KUKA KRL program: ho_lca_st03_pos03.src, ho_lca_st03_pos03.dat

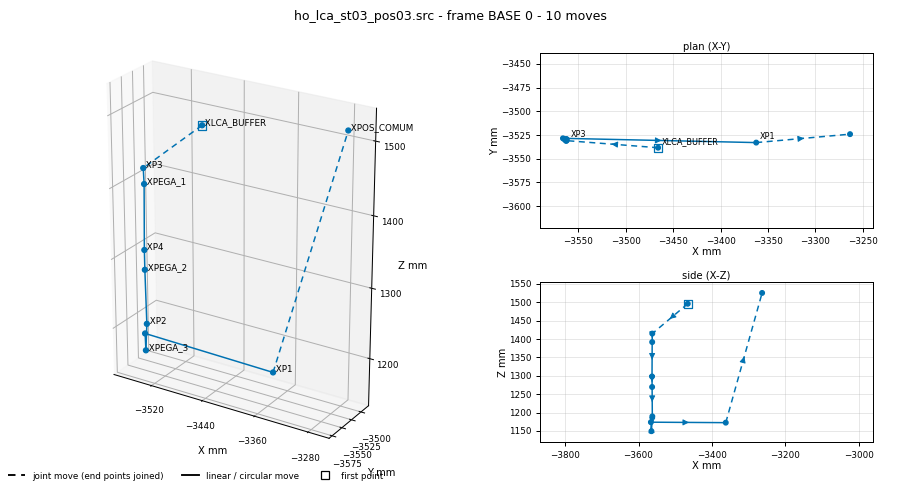
[picture p0: tool path of ho_lca_st03_pos03.src in frame BASE 0, 10 of 10 moves have a stored position in this frame; points joined in program order, loops and branches not executed]
--- ho_lca_st03_pos03.src ---
&ACCESS RVP7
&REL 14
&COMMENT POS_3 LCA
&PARAM DISKPATH = KRC:\R1\Program\LCA
&PARAM TEMPLATE = C:\KRC\Roboter\Template\vorgabe
&PARAM EDITMASK = *
DEF ho_lca_st03_pos03( )
;FOLD INI
  ;FOLD BASISTECH INI
    GLOBAL INTERRUPT DECL 3 WHEN $STOPMESS==TRUE DO IR_STOPM ( )
    INTERRUPT ON 3
    BAS (#INITMOV,0 )
  ;ENDFOLD (BASISTECH INI)
;FOLD SPOTTECH INI
USERSPOT(#INIT)
;ENDFOLD (SPOTTECH INI)
;FOLD GRIPPERTECH INI
USER_GRP(0,DUMMY,DUMMY,GDEFAULT)
;ENDFOLD (GRIPPERTECH INI)
  ;FOLD USER INI
    ;Make your modifications here

  ;ENDFOLD (USER INI)
;ENDFOLD (INI)

; Caracterizacao dos meios de producao
; Changes: Pega LCA Posicao 3 (Pc 3)
; Versao Atual:05/01/2016
; Name: P13.050-R2

chk_w7_wechs_ok ( )   ; CHECK GRIPPER AXOR/ATEGO

;FOLD PTP LCA_BUFFER Vel=100 % DEFAULT Tool[15]:AUX. LCA Base[0];%{PE}%R 8.2.20,%MKUKATPBASIS,%CMOVE,%VPTP,%P 1:PTP, 2:LCA_BUFFER, 3:, 5:100, 7:DEFAULT
$BWDSTART=FALSE
PDAT_ACT=PDEFAULT
FDAT_ACT=FLCA_BUFFER
BAS(#PTP_PARAMS,100)
PTP XLCA_BUFFER
;ENDFOLD

;FOLD WAIT FOR ( IN 3362 'Lib. Pega LCA pos. 3 Axor/Atego' );%{PE}%R 8.2.20,%MKUKATPBASIS,%CEXT_WAIT_FOR,%VEXT_WAIT_FOR,%P 2:, 4:, 5:$IN, 6:3362, 7:Lib. Pega LCA pos. 3 Axor/Atego, 9:
WAIT FOR  ( $IN[3362] )
;ENDFOLD

;FOLD PTP P3 Vel=100 % PDAT1 Tool[15]:AUX. LCA Base[0];%{PE}%R 8.2.20,%MKUKATPBASIS,%CMOVE,%VPTP,%P 1:PTP, 2:P3, 3:, 5:100, 7:PDAT1
$BWDSTART=FALSE
PDAT_ACT=PPDAT1
FDAT_ACT=FP3
BAS(#PTP_PARAMS,100)
PTP XP3
;ENDFOLD

;FOLD WAIT FOR ( NOT IN 489 'Presença pç 1 - Axor LCA' );%{PE}%R 8.2.20,%MKUKATPBASIS,%CEXT_WAIT_FOR,%VEXT_WAIT_FOR,%P 2:, 4:NOT, 5:$IN, 6:489, 7:Presença pç 1 - Axor LCA, 9:
WAIT FOR  (  NOT $IN[489] )
;ENDFOLD

;FOLD ; POSIÇÃO 1 LCA AUSENTE;%{PE}%R 8.2.20,%MKUKATPBASIS,%CCOMMENT,%VNORMAL,%P 2:POSIÇÃO  1 LCA  AUSENTE
;ENDFOLD
;FOLD LIN PEGA_1 Vel=0.1 m/s L_OLP8 Tool[15]:AUX. LCA Base[0];%{PE}%R 8.2.20,%MKUKATPBASIS,%CMOVE,%VLIN,%P 1:LIN, 2:PEGA_1, 3:, 5:0.1, 7:L_OLP8
$BWDSTART=FALSE
LDAT_ACT=LL_OLP8
FDAT_ACT=FPEGA_1
BAS(#CP_PARAMS,0.1)
LIN XPEGA_1
;ENDFOLD

;FOLD LIN P4 Vel=0.05 m/s CPDAT3 Tool[15]:AUX. LCA Base[0];%{PE}%R 8.2.20,%MKUKATPBASIS,%CMOVE,%VLIN,%P 1:LIN, 2:P4, 3:, 5:0.05, 7:CPDAT3
$BWDSTART=FALSE
LDAT_ACT=LCPDAT3
FDAT_ACT=FP4
BAS(#CP_PARAMS,0.05)
LIN XP4
;ENDFOLD

;FOLD WAIT FOR ( NOT IN 489 'Presença pç 1 - Axor LCA' );%{PE}%R 8.2.20,%MKUKATPBASIS,%CEXT_WAIT_FOR,%VEXT_WAIT_FOR,%P 2:, 4:NOT, 5:$IN, 6:489, 7:Presença pç 1 - Axor LCA, 9:
WAIT FOR  (  NOT $IN[489] )
;ENDFOLD

;FOLD ; POSIÇÃO 2 LCA AUSENTE;%{PE}%R 8.2.20,%MKUKATPBASIS,%CCOMMENT,%VNORMAL,%P 2:POSIÇÃO  2 LCA  AUSENTE
;ENDFOLD
;FOLD LIN PEGA_2 Vel=0.05 m/s L_OLP7 Tool[15]:AUX. LCA Base[0];%{PE}%R 8.2.20,%MKUKATPBASIS,%CMOVE,%VLIN,%P 1:LIN, 2:PEGA_2, 3:, 5:0.05, 7:L_OLP7
$BWDSTART=FALSE
LDAT_ACT=LL_OLP7
FDAT_ACT=FPEGA_2
BAS(#CP_PARAMS,0.05)
LIN XPEGA_2
;ENDFOLD

;FOLD LIN P2 Vel=0.05 m/s CPDAT2 Tool[15]:AUX. LCA Base[0];%{PE}%R 8.2.20,%MKUKATPBASIS,%CMOVE,%VLIN,%P 1:LIN, 2:P2, 3:, 5:0.05, 7:CPDAT2
$BWDSTART=FALSE
LDAT_ACT=LCPDAT2
FDAT_ACT=FP2
BAS(#CP_PARAMS,0.05)
LIN XP2
;ENDFOLD

;FOLD ; POSIÇÃO 3 DE PEGA DA PEÇA;%{PE}%R 8.2.20,%MKUKATPBASIS,%CCOMMENT,%VNORMAL,%P 2:POSIÇÃO  3 DE PEGA DA PEÇA
;ENDFOLD
;FOLD LIN PEGA_3 Vel=0.05 m/s L_OLP5 Tool[15]:AUX. LCA Base[0];%{PE}%R 8.2.20,%MKUKATPBASIS,%CMOVE,%VLIN,%P 1:LIN, 2:PEGA_3, 3:, 5:0.05, 7:L_OLP5
$BWDSTART=FALSE
LDAT_ACT=LL_OLP5
FDAT_ACT=FPEGA_3
BAS(#CP_PARAMS,0.05)
LIN XPEGA_3
;ENDFOLD

IF (NOT(GHOST())) THEN
;FOLD WAIT FOR ( IN 489 'Presença pç 1 - Axor LCA' );%{PE}%R 8.2.20,%MKUKATPBASIS,%CEXT_WAIT_FOR,%VEXT_WAIT_FOR,%P 2:, 4:, 5:$IN, 6:489, 7:Presença pç 1 - Axor LCA, 9:
WAIT FOR  ( $IN[489] )
;ENDFOLD
ENDIF

;FOLD SET Z4.1 GRP AXOR State= GDAT7;%{PE}%R 8.2.1,%MKUKATPGRP,%CGRP,%VGRP,%P 2:12, 4:2, 5:#NO, 6:GDAT7, 8:0, 10:0
H50(GRP,12,2,GGDAT7)
;ENDFOLD
chk_w7_grp4_clo()

IF (NOT(GHOST())) THEN
;FOLD SET VACUO AXOR State= GDAT5;%{PE}%R 8.2.1,%MKUKATPGRP,%CGRP,%VGRP,%P 2:9, 4:1, 5:#NO, 6:GDAT5, 8:0, 10:0
H50(GRP,9,1,GGDAT5)
;ENDFOLD
chk_w7_grp1_vac()
ENDIF

;FOLD OUT 3371 'Lib. p/ sair c/ Travessa Axor/Atego' State=TRUE ;%{PE}%R 8.2.20,%MKUKATPBASIS,%COUT,%VOUTX,%P 2:3371, 3:Lib. p/ sair c/ Travessa Axor/Atego, 5:TRUE, 6:
$OUT[3371]=TRUE
;ENDFOLD
;FOLD WAIT Time=1 sec;%{PE}%R 8.2.20,%MKUKATPBASIS,%CWAIT,%VWAIT,%P 3:1
WAIT SEC 1
;ENDFOLD
;FOLD WAIT FOR ( IN 3371 'Lib. p/ Sair c/ Pç LCA Axor/Atego' );%{PE}%R 8.2.20,%MKUKATPBASIS,%CEXT_WAIT_FOR,%VEXT_WAIT_FOR,%P 2:, 4:, 5:$IN, 6:3371, 7:Lib. p/ Sair c/ Pç LCA Axor/Atego, 9:
WAIT FOR  ( $IN[3371] )
;ENDFOLD
;FOLD OUT 3371 'Lib. p/ sair c/ Travessa Axor/Atego' State=FALSE ;%{PE}%R 8.2.20,%MKUKATPBASIS,%COUT,%VOUTX,%P 2:3371, 3:Lib. p/ sair c/ Travessa Axor/Atego, 5:FALSE, 6:
$OUT[3371]=FALSE
;ENDFOLD
;FOLD OUT 3349 'R2 pegou peça' State=FALSE ;%{PE}%R 8.2.20,%MKUKATPBASIS,%COUT,%VOUTX,%P 2:3349, 3:R2 pegou peça, 5:FALSE, 6:
$OUT[3349]=FALSE
;ENDFOLD

;FOLD LIN l040 Vel=0.05 m/s L_OLP6 Tool[15]:AUX. LCA Base[0];%{PE}%R 8.2.20,%MKUKATPBASIS,%CMOVE,%VLIN,%P 1:LIN, 2:l040, 3:, 5:0.05, 7:L_OLP6
$BWDSTART=FALSE
LDAT_ACT=LL_OLP6
FDAT_ACT=Fl040
BAS(#CP_PARAMS,0.05)
LIN Xl040
;ENDFOLD

IF (NOT(GHOST())) THEN
;FOLD WAIT FOR ( IN 489 'Presença pç 1 - Axor LCA' );%{PE}%R 8.2.20,%MKUKATPBASIS,%CEXT_WAIT_FOR,%VEXT_WAIT_FOR,%P 2:, 4:, 5:$IN, 6:489, 7:Presença pç 1 - Axor LCA, 9:
WAIT FOR  ( $IN[489] )
;ENDFOLD
ENDIF

;FOLD LIN P1 Vel=0.05 m/s CPDAT1 Tool[15]:AUX. LCA Base[0];%{PE}%R 8.2.20,%MKUKATPBASIS,%CMOVE,%VLIN,%P 1:LIN, 2:P1, 3:, 5:0.05, 7:CPDAT1
$BWDSTART=FALSE
LDAT_ACT=LCPDAT1
FDAT_ACT=FP1
BAS(#CP_PARAMS,0.05)
LIN XP1
;ENDFOLD

;FOLD ; POSIÇÃO COMUM;%{PE}%R 8.2.20,%MKUKATPBASIS,%CCOMMENT,%VNORMAL,%P 2:POSIÇÃO COMUM
;ENDFOLD
;FOLD PTP POS_COMUM Vel=100 % PDAT0 Tool[15]:AUX. LCA Base[0];%{PE}%R 8.2.20,%MKUKATPBASIS,%CMOVE,%VPTP,%P 1:PTP, 2:POS_COMUM, 3:, 5:100, 7:PDAT0
$BWDSTART=FALSE
PDAT_ACT=PPDAT0
FDAT_ACT=FPOS_COMUM
BAS(#PTP_PARAMS,100)
PTP XPOS_COMUM
;ENDFOLD

END

--- ho_lca_st03_pos03.dat ---
&ACCESS RVP7
&REL 14
&COMMENT POS_3 LCA
&PARAM DISKPATH = KRC:\R1\Program\LCA
&PARAM TEMPLATE = C:\KRC\Roboter\Template\vorgabe
&PARAM EDITMASK = *
DEFDAT  ho_lca_st03_pos03
;FOLD EXTERNAL DECLARATIONS;%{PE}%MKUKATPBASIS,%CEXT,%VCOMMON,%P
;FOLD GRIPPERTECH EXT
EXT  H50 (INT  :IN,INT  :IN,INT  :IN,GRP_TYP  :IN )
;ENDFOLD (GRIPPERTECH EXT)
;FOLD SPOTTECH EXT
EXT  USERSPOT (S_COMMAND  :IN,SPOT_TYPE  :IN )
;ENDFOLD (SPOTTECH EXT)
;FOLD BASISTECH EXT;%{PE}%MKUKATPBASIS,%CEXT,%VEXT,%P
EXT  BAS (BAS_COMMAND  :IN,REAL  :IN )
DECL INT SUCCESS
;ENDFOLD (BASISTECH EXT)
;FOLD USER EXT;%{E}%MKUKATPUSER,%CEXT,%VEXT,%P
;Make your modifications here

;ENDFOLD (USER EXT)
;ENDFOLD (EXTERNAL DECLARATIONS)
DECL BASIS_SUGG_T LAST_BASIS={POINT1[] "P4                      ",POINT2[] "P4                      ",CP_PARAMS[] "CPDAT3                  ",PTP_PARAMS[] "PDAT1                   ",CONT[] "                        ",CP_VEL[] "0.05                    ",PTP_VEL[] "100                     ",SYNC_PARAMS[] "SYNCDAT                 ",SPL_NAME[] "S0                      "}
DECL LDAT LL_OLP5={VEL 0.25,ACC 100.0,APO_DIST 0.0,APO_FAC 0.0,ORI_TYP #VAR,CIRC_TYP #BASE,JERK_FAC 50.0}
DECL GRP_SUGG_T LAST_GRP={NUMBER[] "9                       ",STATE[] "1                       ",PARAMS[] "GDAT1                   "}
DECL GRP_TYP GGDAT6={G_APO #NO,GRP_TIME 0.200000003,CTRL #OFF,DLY 0,DST 1}
DECL LDAT LL_OLP6={VEL 0.25,ACC 100.0,APO_DIST 0.0,APO_FAC 0.0,ORI_TYP #VAR,CIRC_TYP #BASE,JERK_FAC 50.0}
DECL E6POS Xl040={X -3566.28296,Y -3528.49805,Z 1173.75195,A -1.25957894,B 0.337334186,C -176.389099,S 6,T 26,E1 -3443.72803,E2 0.0,E3 0.0,E4 0.0,E5 0.0,E6 0.0}
DECL FDAT Fl040={TOOL_NO 15,BASE_NO 0,IPO_FRAME #BASE,POINT2[] " ",TQ_STATE FALSE}
DECL GRP_TYP GGDAT1={G_APO #NO,GRP_TIME 0.200000003,CTRL #OFF,DLY 0,DST 1}
DECL GRP_TYP GGDAT2={G_APO #NO,GRP_TIME 0.200000003,CTRL #OFF,DLY 0,DST 1}
DECL PDAT PPDAT0={VEL 100.0,ACC 100.0,APO_DIST 100.0}
DECL E6POS XPOS_COMUM={X -3263.56592,Y -3524.10889,Z 1525.54504,A 0.586738884,B -3.95688391,C -178.223694,S 6,T 26,E1 -3443.7251,E2 0.0,E3 0.0,E4 0.0,E5 0.0,E6 0.0}
DECL FDAT FPOS_COMUM={TOOL_NO 15,BASE_NO 0,IPO_FRAME #BASE,POINT2[] " ",TQ_STATE FALSE}
DECL GRP_TYP GGDAT3={G_APO #NO,GRP_TIME 0.200000003,CTRL #OFF,DLY 0,DST 1}
DECL GRP_TYP GGDAT4={G_APO #NO,GRP_TIME 0.200000003,CTRL #OFF,DLY 0,DST 1}
DECL E6POS XP1={X -3362.49609,Y -3533.0,Z 1172.49597,A -1.25867605,B 0.334295392,C -176.389893,S 6,T 26,E1 -3443.729,E2 0.0,E3 0.0,E4 0.0,E5 0.0,E6 0.0}
DECL FDAT FP1={TOOL_NO 15,BASE_NO 0,IPO_FRAME #BASE,POINT2[] " ",TQ_STATE FALSE}
DECL LDAT LCPDAT1={VEL 2.0,ACC 100.0,APO_DIST 100.0,APO_FAC 50.0,AXIS_VEL 100.0,AXIS_ACC 100.0,ORI_TYP #VAR,CIRC_TYP #BASE,JERK_FAC 50.0,GEAR_JERK 50.0,EXAX_IGN 0}
DECL GRP_TYP GGDAT7={G_APO #NO,GRP_TIME 0.200000003,CTRL #OFF,DLY 0,DST 1}
DECL GRP_TYP GGDAT5={G_APO #NO,GRP_TIME 0.200000003,CTRL #OFF,DLY 0,DST 1}
DECL E6POS XLCA_BUFFER={X -3465.96704,Y -3538.40991,Z 1496.08801,A -1.25961006,B 0.337735415,C -176.389206,S 6,T 26,E1 -3443.72705,E2 0.0,E3 0.0,E4 0.0,E5 0.0,E6 0.0}
DECL FDAT FLCA_BUFFER={TOOL_NO 15,BASE_NO 0,IPO_FRAME #BASE,POINT2[] " ",TQ_STATE FALSE}
DECL E6POS XP2={X -3562.38208,Y -3529.57495,Z 1189.53101,A -1.25961101,B 0.337735415,C -176.389206,S 6,T 26,E1 -3443.72705,E2 0.0,E3 0.0,E4 0.0,E5 0.0,E6 0.0}
DECL FDAT FP2={TOOL_NO 15,BASE_NO 0,IPO_FRAME #BASE,POINT2[] " ",TQ_STATE FALSE}
DECL LDAT LCPDAT2={VEL 2.0,ACC 100.0,APO_DIST 100.0,APO_FAC 50.0,AXIS_VEL 100.0,AXIS_ACC 100.0,ORI_TYP #VAR,CIRC_TYP #BASE,JERK_FAC 50.0,GEAR_JERK 50.0,EXAX_IGN 0}
DECL E6POS XPEGA_5={X -3564.81592,Y -3529.46899,Z 1149.26904,A -1.25961006,B 0.337735295,C -176.389206,S 6,T 26,E1 -3443.72705,E2 0.0,E3 0.0,E4 0.0,E5 0.0,E6 0.0}
DECL FDAT FPEGA_5={TOOL_NO 15,BASE_NO 0,IPO_FRAME #BASE,POINT2[] " ",TQ_STATE FALSE}
DECL E6POS XPEGA_3={X -3564.80811,Y -3529.4729,Z 1149.23096,A -1.25936401,B 0.335955292,C -176.389206,S 6,T 26,E1 -3443.72705,E2 0.0,E3 0.0,E4 0.0,E5 0.0,E6 0.0}
DECL FDAT FPEGA_3={TOOL_NO 15,BASE_NO 0,IPO_FRAME #BASE,POINT2[] " ",TQ_STATE FALSE}
DECL LDAT LL_OLP7={VEL 0.25,ACC 100.0,APO_DIST 0.0,APO_FAC 0.0,ORI_TYP #VAR,CIRC_TYP #BASE,JERK_FAC 50.0}
DECL E6POS XPEGA_2={X -3562.96509,Y -3530.99512,Z 1269.58606,A -1.25582802,B 0.336914808,C -176.399597,S 6,T 26,E1 -3443.72803,E2 0.0,E3 0.0,E4 0.0,E5 0.0,E6 0.0}
DECL FDAT FPEGA_2={TOOL_NO 15,BASE_NO 0,IPO_FRAME #BASE,POINT2[] " ",TQ_STATE FALSE}
DECL LDAT LL_OLP8={VEL 0.25,ACC 100.0,APO_DIST 0.0,APO_FAC 0.0,ORI_TYP #VAR,CIRC_TYP #BASE,JERK_FAC 50.0}
DECL E6POS XPEGA_1={X -3562.76904,Y -3529.24512,Z 1391.84998,A -1.43793905,B 0.495635509,C -176.2565,S 6,T 26,E1 -3443.72705,E2 0.0,E3 0.0,E4 0.0,E5 0.0,E6 0.0}
DECL FDAT FPEGA_1={TOOL_NO 15,BASE_NO 0,IPO_FRAME #BASE,POINT2[] " ",TQ_STATE FALSE}
DECL PDAT PPDAT1={VEL 100.0,ACC 100.0,APO_DIST 100.0}
DECL E6POS XP3={X -3562.46509,Y -3530.94409,Z 1414.94702,A -1.32614005,B 0.398220807,C -176.339493,S 6,T 26,E1 -3443.72803,E2 0.0,E3 0.0,E4 0.0,E5 0.0,E6 0.0}
DECL FDAT FP3={TOOL_NO 15,BASE_NO 0,IPO_FRAME #BASE,POINT2[] " ",TQ_STATE FALSE}
DECL LDAT LCPDAT3={VEL 2.0,ACC 100.0,APO_DIST 100.0,APO_FAC 50.0,AXIS_VEL 100.0,AXIS_ACC 100.0,ORI_TYP #VAR,CIRC_TYP #BASE,JERK_FAC 50.0,GEAR_JERK 50.0,EXAX_IGN 0}
DECL E6POS XP4={X -3563.21191,Y -3530.92212,Z 1298.24097,A -1.258762,B 0.337085485,C -176.391403,S 6,T 26,E1 -3443.72705,E2 0.0,E3 0.0,E4 0.0,E5 0.0,E6 0.0}
DECL FDAT FP4={TOOL_NO 15,BASE_NO 0,IPO_FRAME #BASE,POINT2[] " ",TQ_STATE FALSE}
ENDDAT
